(* IEC 61131-3 sources: crb-codesys/generation/scripts/repoeval/PID_controller/Globals, 3 files *)

(* ---- GVL_Input.st ---- *)
VAR_GLOBAL
	Knapp1: BOOL; // Knapp på våning 1
	Knapp2: BOOL; //
	Knapp3: BOOL;
	Knapp4: BOOL;
	Vaning1 :BOOL;
	Vaning2 :BOOL;
	Vaning3 :BOOL;
	Vaning4 :BOOL;
	Manuell :BOOL;
	Auto :BOOL;
	Upp :BOOL;
	Ner  :BOOL;
	Service_reset :BOOL;
END_VAR

(* ---- GVL_Memory.st ---- *)
VAR_GLOBAL
END_VAR

(* ---- GVL_Output.st ---- *)
VAR_GLOBAL
	Lampa1 :BOOL;
	Lampa2 :BOOL;
	Lampa3 :BOOL;
	Lampa4 :BOOL;
	HissUpp :BOOL;
	HissNer :BOOL;
	HissDorr :BOOL;
	LampaAuto :BOOL;

END_VAR
